FUNCTION Convert_UDINT_TO_DINT : Hresult
VAR_INPUT
	in : UDINT;
	out : REFERENCE TO DINT;
END_VAR
VAR
	converted : DINT;
END_VAR
VAR CONSTANT
	INCOMPATIBLE : HRESULT := 16#9811070E;
END_VAR

converted := UDINT_TO_DINT(in);

IF (DINT_TO_UDINT(converted) <> in) THEN
	Convert_UDINT_TO_DINT := INCOMPATIBLE;
	RETURN;
END_IF

out := converted;

END_FUNCTION

(* stored: Version 1.1.0.1, ProductVersion 3.1.4024.12
   POU Convert_UDINT_TO_DINT: Id {45be4b51-4b0a-401a-9cec-c9ae4dcb11aa}, SpecialFunc None *)
